INTERFACE IPicker EXTENDS ZApplication.IUnit

END_INTERFACE

(* stored: Version 1.1.0.1
   Itf IPicker: Id {f87da058-7205-4724-9451-f3d4174d563f} *)
